TYPE stNested :
STRUCT
	{attribute addProperty Name "Name"}
	Name : STRING;
	{attribute addProperty Name "Turn on nested station"}
	NestedOn : BOOL;	
	{attribute addProperty Name "Date and Time"}
	TestDateTime : DATE_AND_TIME;	
END_STRUCT
END_TYPE

(* stored: Version 1.1.0.1, ProductVersion 3.1.4024.6
   DUT stNested: Id {aa801c5f-eb15-0419-0182-555df9d9606c} *)
